// TIA Portal project "PROJEKT_PLC_PALIWKO" (V15.1)

(* hardware
DEVICE "S7-1200 station_1"  S7-1200 Station
   slot 0: "Rack_0"  S7-1200 Rack  Rack  V1.0
   slot 1: "PLC_1"  CPU 1212C AC/DC/Rly  6ES7 212-1BE40-0XB0  V4.2
DEVICE "HMI_1"  KTP700 Basic PN
   slot 0: "HMI_1"  KTP700 Basic PN  6AV2 123-2GB03-0AX0  15.0.0.0
   slot 1: "HMI_RT_1"  KTP700 Basic PN  6AV2 123-2GB03-0AX0  15.0.0.0
   slot 5: "HMI_1.IE_CP_1"  PROFINET Interface  15.0.0.0
      slot 1: "PROFINET Interface_1"  PROFINET Interface
         slot 1: "Port_1"  Port
*)

// ===== PLC "PLC_1"  CPU 1212C AC/DC/Rly =====

VAR_GLOBAL   // PLC tag table "Default tag table"
   "Adam" AT %M0.1 : Bool;
   "Ignacy" AT %M0.2 : Bool;
   "Kuba" AT %M0.3 : Bool;
   "Mateusz" AT %M0.4 : Bool;
   "Stachu" AT %M0.5 : Bool;
   "Limit_paliwa_adam" AT %M10.0 : Bool;
   "Limit_paliwa_ignacy" AT %M10.2 : Bool;
   "Limit_paliwa_kuba" AT %M10.3 : Bool;
   "Limit_paliwa_stachu" AT %M10.4 : Bool;
   "Limit_paliwa_mateusz" AT %M10.5 : Bool;
   "FuelingActive" AT %M10.6 : Bool;
   "Blokada_nalewania1" AT %M100.1 : Bool;
   "Blokada_nalewania2" AT %M100.2 : Bool;
   "Blokada_przelania_adam" AT %M4.0 : Bool;
   "Blokada_przelania_ignacy" AT %M4.1 : Bool;
   "Blokada_przelania_kuba" AT %M4.2 : Bool;
   "Blokada_przelania_mateusz" AT %M4.3 : Bool;
   "Blokada_przelania_stachu" AT %M4.4 : Bool;
END_VAR

TYPE "Kierowca"
   STRUCT
      Imie : String;
      Ilosc_Paliwa_Z : Int;
      Data_wydania : DTL;
   END_STRUCT;
END_TYPE

DATA_BLOCK "User_Data"   // DB1
{ S7_Optimized_Access := 'TRUE' }
VERSION : 0.1
   VAR
      Login : String;
      Adam : "Kierowca";
      Kuba : "Kierowca";
      Stachu : "Kierowca";
      Ignacy : "Kierowca";
      Mateusz : "Kierowca";
      Czy_Nalac : Bool;
      Done : Int;
   END_VAR
BEGIN
   Adam.Ilosc_Paliwa_Z := 200;
   Adam.Imie := 'Adam';
   Kuba.Imie := 'Kuba';
   Kuba.Ilosc_Paliwa_Z := 200;
   Stachu.Imie := 'Stachu';
   Stachu.Ilosc_Paliwa_Z := 200;
   Ignacy.Imie := 'Ignacy';
   Ignacy.Ilosc_Paliwa_Z := 200;
   Mateusz.Imie := 'Mateusz';
   Mateusz.Ilosc_Paliwa_Z := 200;
END_DATA_BLOCK

DATA_BLOCK "HMI"   // DB2
{ S7_Optimized_Access := 'TRUE' }
VERSION : 0.1
   VAR
      Current_User : String;
      Godzina : Time_Of_Day;
      Data : Date;
      Ile_Paliwa_z : Int;
      Ile_Paliwa_n : Int;
      Czy_nalac : Bool;
      Nalewanie_aktywne : Bool;
   END_VAR
BEGIN
END_DATA_BLOCK

DATA_BLOCK "Block_1_DB"   // DB3
{ S7_Optimized_Access := 'TRUE' }
VERSION : 0.1
// stored: InstanceOfName Block_1
"Block_1"
BEGIN
END_DATA_BLOCK

// folder: System blocks/Program resources

DATA_BLOCK "IEC_Timer_0_DB"   // DB5
{ S7_Optimized_Access := 'TRUE' }
AUTHOR : Simatic
FAMILY : IEC
NAME : IEC_TMR
VERSION : 1.0
// stored: InstanceOfName IEC_TIMER
"IEC_TIMER"
BEGIN
END_DATA_BLOCK

DATA_BLOCK "IEC_Timer_0_DB_1"   // DB6
{ S7_Optimized_Access := 'TRUE' }
AUTHOR : Simatic
FAMILY : IEC
NAME : IEC_TMR
VERSION : 1.0
// stored: InstanceOfName IEC_TIMER
"IEC_TIMER"
BEGIN
END_DATA_BLOCK

// folder: (top level)

FUNCTION_BLOCK "Block_1"   // FB1, LAD
TITLE = Pouring
{ S7_Optimized_Access := 'TRUE' }
VERSION : 0.1
// All the fuel dispensing logic happens
   VAR_TEMP   // added for the SCL form of the ladder/FBD networks
      _w1 : Bool;
   END_VAR
BEGIN

REGION Network 1: Trigger
   // Triggering the "pour" sequence
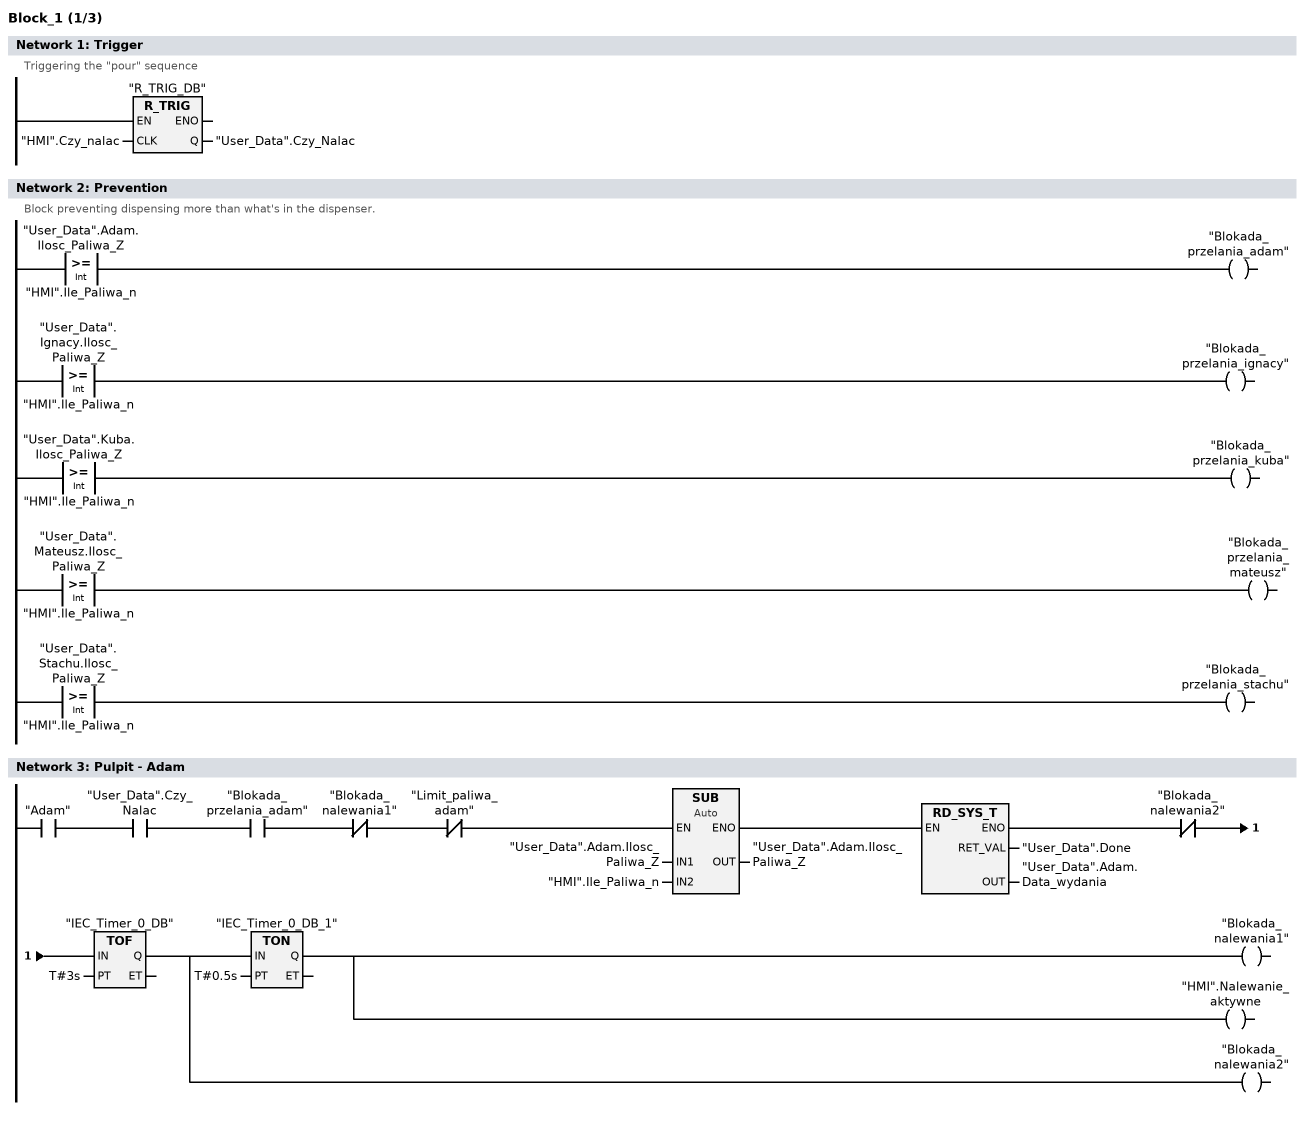
   "R_TRIG_DB"(CLK := "HMI".Czy_nalac, Q => "User_Data".Czy_Nalac);   // R_TRIG
END_REGION

REGION Network 2: Prevention
   // Block preventing dispensing more than what's in the dispenser.
   RUNG wire#powerrail
      { S7_Templates := "SrcType := Int" } GE_Contact(in1 := "User_Data".Adam.Ilosc_Paliwa_Z, in2 := "HMI".Ile_Paliwa_n)
      Coil( "Blokada_przelania_adam" )
   END_RUNG
   RUNG wire#powerrail
      { S7_Templates := "SrcType := Int" } GE_Contact(in1 := "User_Data".Ignacy.Ilosc_Paliwa_Z, in2 := "HMI".Ile_Paliwa_n)
      Coil( "Blokada_przelania_ignacy" )
   END_RUNG
   RUNG wire#powerrail
      { S7_Templates := "SrcType := Int" } GE_Contact(in1 := "User_Data".Kuba.Ilosc_Paliwa_Z, in2 := "HMI".Ile_Paliwa_n)
      Coil( "Blokada_przelania_kuba" )
   END_RUNG
   RUNG wire#powerrail
      { S7_Templates := "SrcType := Int" } GE_Contact(in1 := "User_Data".Mateusz.Ilosc_Paliwa_Z, in2 := "HMI".Ile_Paliwa_n)
      Coil( "Blokada_przelania_mateusz" )
   END_RUNG
   RUNG wire#powerrail
      { S7_Templates := "SrcType := Int" } GE_Contact(in1 := "User_Data".Stachu.Ilosc_Paliwa_Z, in2 := "HMI".Ile_Paliwa_n)
      Coil( "Blokada_przelania_stachu" )
   END_RUNG
   // the same network as SCL:
   "Blokada_przelania_adam" := "User_Data".Adam.Ilosc_Paliwa_Z >= "HMI".Ile_Paliwa_n;
   "Blokada_przelania_ignacy" := "User_Data".Ignacy.Ilosc_Paliwa_Z >= "HMI".Ile_Paliwa_n;
   "Blokada_przelania_kuba" := "User_Data".Kuba.Ilosc_Paliwa_Z >= "HMI".Ile_Paliwa_n;
   "Blokada_przelania_mateusz" := "User_Data".Mateusz.Ilosc_Paliwa_Z >= "HMI".Ile_Paliwa_n;
   "Blokada_przelania_stachu" := "User_Data".Stachu.Ilosc_Paliwa_Z >= "HMI".Ile_Paliwa_n;
END_REGION

REGION Network 3: Pulpit - Adam
   // ENO of a box is taken as its EN; it also drops when the box reports an error
   #_w1 := "Adam" AND "User_Data".Czy_Nalac AND "Blokada_przelania_adam" AND NOT "Blokada_nalewania1" AND NOT "Limit_paliwa_adam";
   IF #_w1 THEN
       "User_Data".Adam.Ilosc_Paliwa_Z := "User_Data".Adam.Ilosc_Paliwa_Z - "HMI".Ile_Paliwa_n;
       "User_Data".Done := RD_SYS_T(OUT => "User_Data".Adam.Data_wydania);
   END_IF;
   "IEC_Timer_0_DB".TOF(IN := #_w1 AND NOT "Blokada_nalewania2", PT := T#3s);
   "IEC_Timer_0_DB_1".TON(IN := "IEC_Timer_0_DB".Q, PT := T#0.5s);
   "Blokada_nalewania1" := "IEC_Timer_0_DB_1".Q;
   "HMI".Nalewanie_aktywne := "IEC_Timer_0_DB_1".Q;
   "Blokada_nalewania2" := "IEC_Timer_0_DB".Q;
END_REGION

REGION Network 4: Pulpit - Ignacy
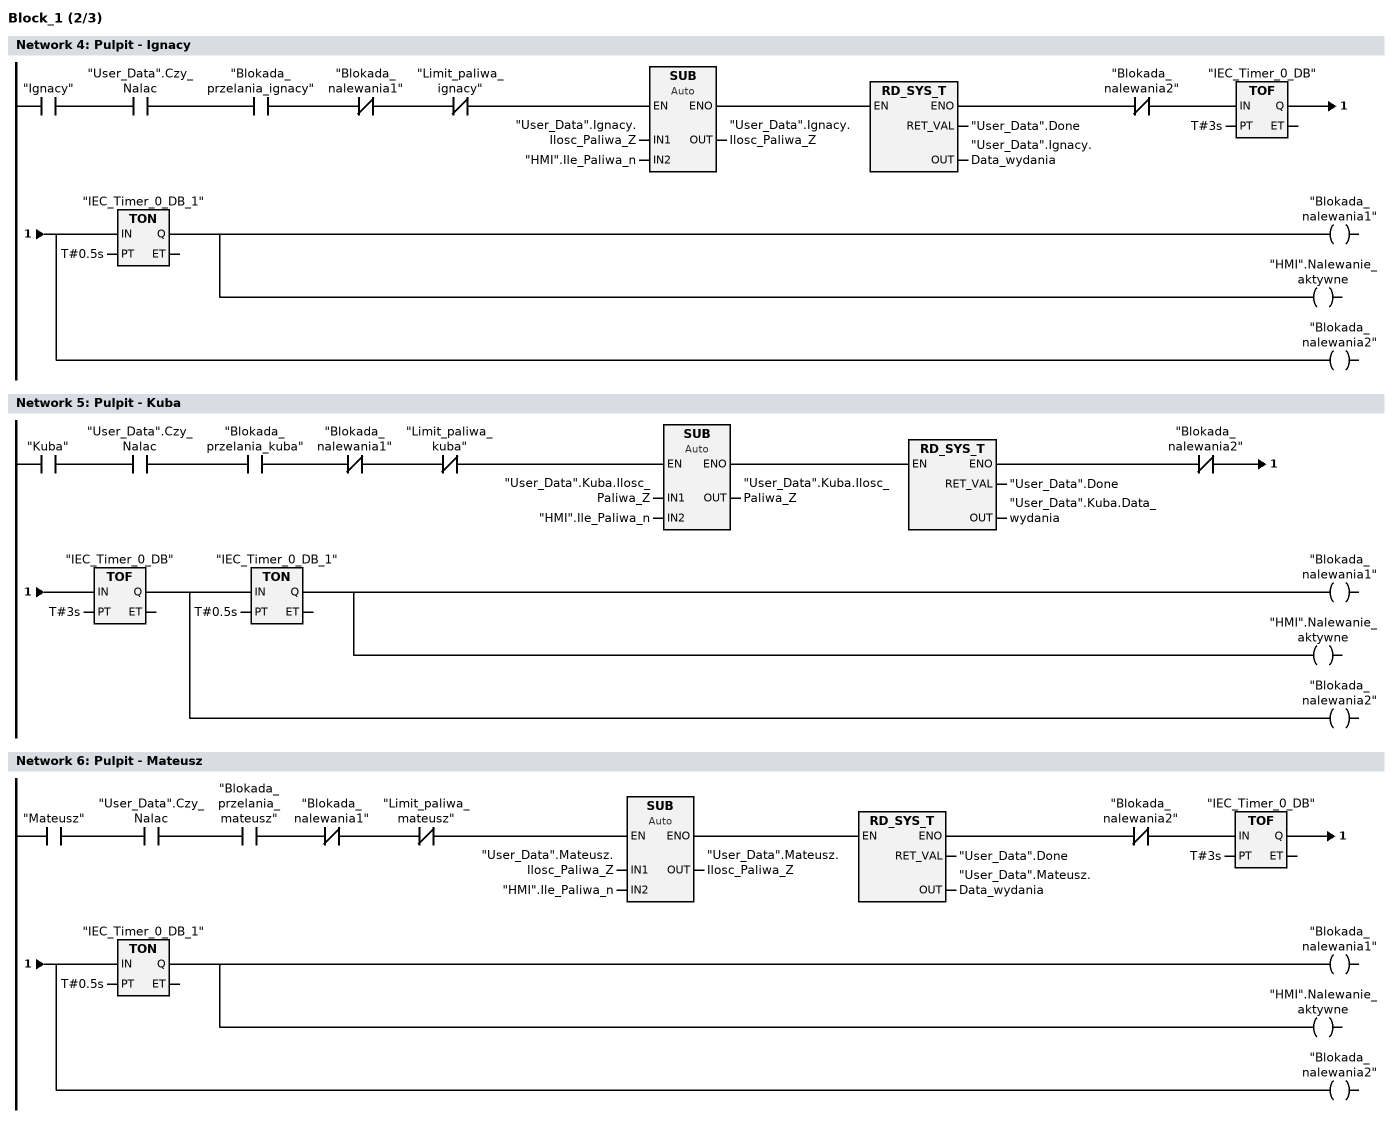
   // ENO of a box is taken as its EN; it also drops when the box reports an error
   #_w1 := "Ignacy" AND "User_Data".Czy_Nalac AND "Blokada_przelania_ignacy" AND NOT "Blokada_nalewania1" AND NOT "Limit_paliwa_ignacy";
   IF #_w1 THEN
       "User_Data".Ignacy.Ilosc_Paliwa_Z := "User_Data".Ignacy.Ilosc_Paliwa_Z - "HMI".Ile_Paliwa_n;
       "User_Data".Done := RD_SYS_T(OUT => "User_Data".Ignacy.Data_wydania);
   END_IF;
   "IEC_Timer_0_DB".TOF(IN := #_w1 AND NOT "Blokada_nalewania2", PT := T#3s);
   "IEC_Timer_0_DB_1".TON(IN := "IEC_Timer_0_DB".Q, PT := T#0.5s);
   "Blokada_nalewania1" := "IEC_Timer_0_DB_1".Q;
   "HMI".Nalewanie_aktywne := "IEC_Timer_0_DB_1".Q;
   "Blokada_nalewania2" := "IEC_Timer_0_DB".Q;
END_REGION

REGION Network 5: Pulpit - Kuba
   // ENO of a box is taken as its EN; it also drops when the box reports an error
   #_w1 := "Kuba" AND "User_Data".Czy_Nalac AND "Blokada_przelania_kuba" AND NOT "Blokada_nalewania1" AND NOT "Limit_paliwa_kuba";
   IF #_w1 THEN
       "User_Data".Kuba.Ilosc_Paliwa_Z := "User_Data".Kuba.Ilosc_Paliwa_Z - "HMI".Ile_Paliwa_n;
       "User_Data".Done := RD_SYS_T(OUT => "User_Data".Kuba.Data_wydania);
   END_IF;
   "IEC_Timer_0_DB".TOF(IN := #_w1 AND NOT "Blokada_nalewania2", PT := T#3s);
   "IEC_Timer_0_DB_1".TON(IN := "IEC_Timer_0_DB".Q, PT := T#0.5s);
   "Blokada_nalewania1" := "IEC_Timer_0_DB_1".Q;
   "HMI".Nalewanie_aktywne := "IEC_Timer_0_DB_1".Q;
   "Blokada_nalewania2" := "IEC_Timer_0_DB".Q;
END_REGION

REGION Network 6: Pulpit - Mateusz
   // ENO of a box is taken as its EN; it also drops when the box reports an error
   #_w1 := "Mateusz" AND "User_Data".Czy_Nalac AND "Blokada_przelania_mateusz" AND NOT "Blokada_nalewania1" AND NOT "Limit_paliwa_mateusz";
   IF #_w1 THEN
       "User_Data".Mateusz.Ilosc_Paliwa_Z := "User_Data".Mateusz.Ilosc_Paliwa_Z - "HMI".Ile_Paliwa_n;
       "User_Data".Done := RD_SYS_T(OUT => "User_Data".Mateusz.Data_wydania);
   END_IF;
   "IEC_Timer_0_DB".TOF(IN := #_w1 AND NOT "Blokada_nalewania2", PT := T#3s);
   "IEC_Timer_0_DB_1".TON(IN := "IEC_Timer_0_DB".Q, PT := T#0.5s);
   "Blokada_nalewania1" := "IEC_Timer_0_DB_1".Q;
   "HMI".Nalewanie_aktywne := "IEC_Timer_0_DB_1".Q;
   "Blokada_nalewania2" := "IEC_Timer_0_DB".Q;
END_REGION

REGION Network 7: Pulpit - Stachu
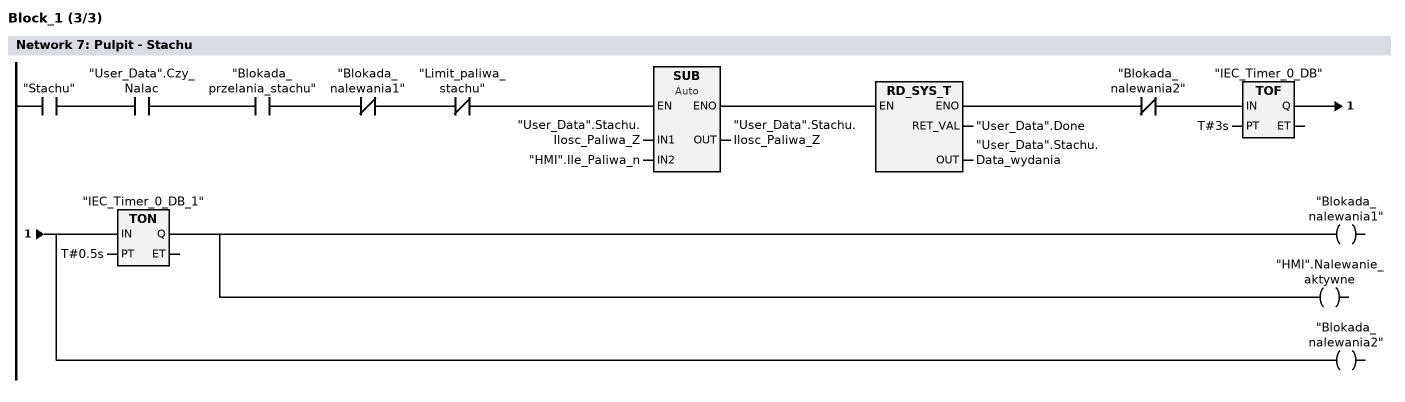
   // ENO of a box is taken as its EN; it also drops when the box reports an error
   #_w1 := "Stachu" AND "User_Data".Czy_Nalac AND "Blokada_przelania_stachu" AND NOT "Blokada_nalewania1" AND NOT "Limit_paliwa_stachu";
   IF #_w1 THEN
       "User_Data".Stachu.Ilosc_Paliwa_Z := "User_Data".Stachu.Ilosc_Paliwa_Z - "HMI".Ile_Paliwa_n;
       "User_Data".Done := RD_SYS_T(OUT => "User_Data".Stachu.Data_wydania);
   END_IF;
   "IEC_Timer_0_DB".TOF(IN := #_w1 AND NOT "Blokada_nalewania2", PT := T#3s);
   "IEC_Timer_0_DB_1".TON(IN := "IEC_Timer_0_DB".Q, PT := T#0.5s);
   "Blokada_nalewania1" := "IEC_Timer_0_DB_1".Q;
   "HMI".Nalewanie_aktywne := "IEC_Timer_0_DB_1".Q;
   "Blokada_nalewania2" := "IEC_Timer_0_DB".Q;
END_REGION
END_FUNCTION_BLOCK

ORGANIZATION_BLOCK "Main"   // OB1, LAD, ProgramCycle
TITLE = "Main Program Sweep (Cycle)"
{ S7_Optimized_Access := 'TRUE' }
VERSION : 0.1
BEGIN

REGION Network 1: User - data
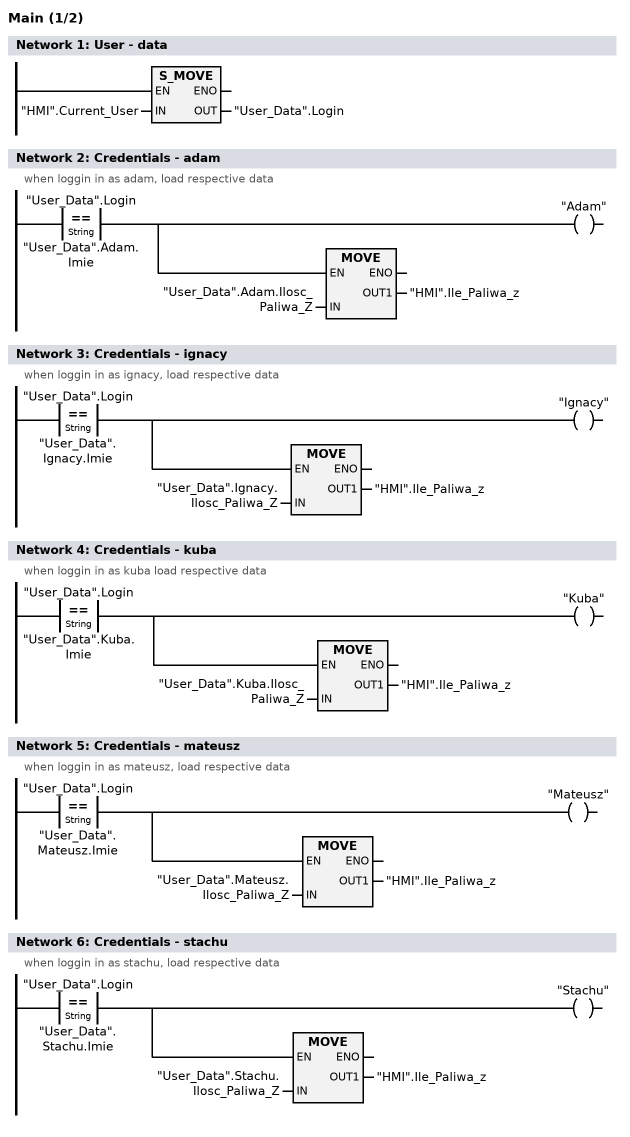
   RUNG wire#powerrail
      S_Move(in := "HMI".Current_User, out => "User_Data".Login)
   END_RUNG
   // the same network as SCL:
   "User_Data".Login := "HMI".Current_User;
END_REGION

REGION Network 2: Credentials - adam
   // when loggin in as adam, load respective data
   RUNG wire#powerrail
      { S7_Templates := "SrcType := String" } EQ_Contact(in1 := "User_Data".Login, in2 := "User_Data".Adam.Imie)
      wire#w1
      Coil( "Adam" )
   END_RUNG
   RUNG wire#w1
      Move(in := "User_Data".Adam.Ilosc_Paliwa_Z, out1 => "HMI".Ile_Paliwa_z)
   END_RUNG
   // the same network as SCL:
   "Adam" := "User_Data".Login = "User_Data".Adam.Imie;
   IF "Adam" THEN "HMI".Ile_Paliwa_z := "User_Data".Adam.Ilosc_Paliwa_Z; END_IF;
END_REGION

REGION Network 3: Credentials - ignacy
   // when loggin in as ignacy, load respective data
   RUNG wire#powerrail
      { S7_Templates := "SrcType := String" } EQ_Contact(in1 := "User_Data".Login, in2 := "User_Data".Ignacy.Imie)
      wire#w1
      Coil( "Ignacy" )
   END_RUNG
   RUNG wire#w1
      Move(in := "User_Data".Ignacy.Ilosc_Paliwa_Z, out1 => "HMI".Ile_Paliwa_z)
   END_RUNG
   // the same network as SCL:
   "Ignacy" := "User_Data".Login = "User_Data".Ignacy.Imie;
   IF "Ignacy" THEN "HMI".Ile_Paliwa_z := "User_Data".Ignacy.Ilosc_Paliwa_Z; END_IF;
END_REGION

REGION Network 4: Credentials - kuba
   // when loggin in as kuba load respective data
   RUNG wire#powerrail
      { S7_Templates := "SrcType := String" } EQ_Contact(in1 := "User_Data".Login, in2 := "User_Data".Kuba.Imie)
      wire#w1
      Coil( "Kuba" )
   END_RUNG
   RUNG wire#w1
      Move(in := "User_Data".Kuba.Ilosc_Paliwa_Z, out1 => "HMI".Ile_Paliwa_z)
   END_RUNG
   // the same network as SCL:
   "Kuba" := "User_Data".Login = "User_Data".Kuba.Imie;
   IF "Kuba" THEN "HMI".Ile_Paliwa_z := "User_Data".Kuba.Ilosc_Paliwa_Z; END_IF;
END_REGION

REGION Network 5: Credentials - mateusz
   // when loggin in as mateusz, load respective data
   RUNG wire#powerrail
      { S7_Templates := "SrcType := String" } EQ_Contact(in1 := "User_Data".Login, in2 := "User_Data".Mateusz.Imie)
      wire#w1
      Coil( "Mateusz" )
   END_RUNG
   RUNG wire#w1
      Move(in := "User_Data".Mateusz.Ilosc_Paliwa_Z, out1 => "HMI".Ile_Paliwa_z)
   END_RUNG
   // the same network as SCL:
   "Mateusz" := "User_Data".Login = "User_Data".Mateusz.Imie;
   IF "Mateusz" THEN "HMI".Ile_Paliwa_z := "User_Data".Mateusz.Ilosc_Paliwa_Z; END_IF;
END_REGION

REGION Network 6: Credentials - stachu
   // when loggin in as stachu, load respective data
   RUNG wire#powerrail
      { S7_Templates := "SrcType := String" } EQ_Contact(in1 := "User_Data".Login, in2 := "User_Data".Stachu.Imie)
      wire#w1
      Coil( "Stachu" )
   END_RUNG
   RUNG wire#w1
      Move(in := "User_Data".Stachu.Ilosc_Paliwa_Z, out1 => "HMI".Ile_Paliwa_z)
   END_RUNG
   // the same network as SCL:
   "Stachu" := "User_Data".Login = "User_Data".Stachu.Imie;
   IF "Stachu" THEN "HMI".Ile_Paliwa_z := "User_Data".Stachu.Ilosc_Paliwa_Z; END_IF;
END_REGION

REGION Network 7: Call FB1
   // FB1 - where all the fuel dispensing logic happens
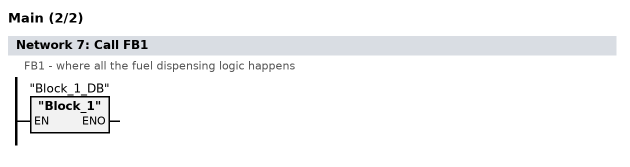
   RUNG wire#powerrail
      "Block_1_DB"()
   END_RUNG
   // the same network as SCL:
   "Block_1_DB"();   // "Block_1"
END_REGION
END_ORGANIZATION_BLOCK

(* ===== HMI "HMI_RT_1" =====
system functions are stored by id; their names below are inferred from use
connection "HMI_Connection_1": ETHERNET, SMART_S7_1200_OMS

HMI tags "Default tag table"
   "HMI_Current_User" : String[254] = PLC HMI.Current_User, 1 s
   "HMI_Ile_Paliwa_z" : Int = PLC HMI.Ile_Paliwa_z, 1 s
   "HMI_Ile_Paliwa_n" : Int = PLC HMI.Ile_Paliwa_n, 1 s
   "HMI_Czy_nalac" : Bool = PLC HMI.Czy_nalac, 1 s
   "HMI_Data_Godzina" : Time_Of_Day = PLC HMI.Godzina, 1 s
   "HMI_Data" : Date = PLC HMI.Data, 1 s
   "HMI_Nalewanie_aktywne" : Bool = PLC HMI.Nalewanie_aktywne AT %DB1.DBX0.0, 500 ms
   "FuelingActive" : Bool = PLC FuelingActive AT %M10.6, 1 s

Template "Template_1" 800x480
   Button "Alarms" at 512,428 size 71x50; TextOff 'Alarms / Alarm'; PictureOff "AlarmDisplay_KTP700_Basic_PN_TR"; PictureOn "AlarmDisplay_KTP700_Basic_PN_TR"
      on Release: function_ef3f5d25("Alarm window_Unacknowledged", -1)
   Button "Exit" at 411,428 size 71x50; TextOff 'Exit'; PictureOff "ExitRuntime_KTP700_Basic_PN_TR"; PictureOn "ExitRuntime_KTP700_Basic_PN_TR"
      on Release: StopRuntime(0)
   Button "Log on" at 311,428 size 71x50; TextOff 'Log on'; PictureOff "Login_KTP700_Basic_PN_TR"; PictureOn "Login_KTP700_Basic_PN_TR"
      on Release: function_a2a04561()
   Button "Start screen" at 211,428 size 71x50; TextOff 'Start screen / Ekran początkowy'; PictureOff "NavigateHome_KTP700_Basic_PN_TR"; PictureOn "NavigateHome_KTP700_Basic_PN_TR"
      on Release: ActivateScreen("Logowanie", 0)

screen "Logowanie" 800x480, template "Template_1"
   on GenerateScreen: function_f41c6f6c("HMI_Current_User")
   Button "Button_1" at 318,194 size 152x88; TextOff 'Log in / Zaloguj / Anmelden'; Authorization "Nalewanie"
      on Click: ActivateScreen("Nalewanie", 0)
   Button "Button_2" at 612,15 size 174x30; TextOff 'Change language / Zmień język / Sprache ändern'
      on Release: function_fb9197e8(-1)
   TextField "Text field_1" at 5,2 size 360x55; Text 'Electronic fuel distribution system / Elektroniczny system rozdzielni paliwa / Elektronisches Kraftstoffverteilungssystem'

screen "Nalewanie" 800x480
   on GenerateScreen: function_f41c6f6c("HMI_Current_User")
   Button "Button_1" at 615,390 size 135x56; TextOff 'Log out / Wyloguj / Abmelden'
      on Click: ActivateScreen("Logowanie", 0); function_f23ef4c9()
   IOField "I/O field_1" at 138,139 size 141x44; FormatPattern s99999
      ProcessValue <- "HMI_Ile_Paliwa_z"
   TextField "Text field_1" at 137,115 size 175x23; Text 'Distributor status / Stan dystrubutora / Status des Verteilers'
   IOField "I/O field_2" at 530,139 size 141x44; FormatPattern s99999
      ProcessValue <- "HMI_Ile_Paliwa_n"
   TextField "Text field_2" at 531,115 size 143x23; Text 'Dispensing order / Zlecenie rozlewu / Abfüllauftrag'
   Button "Button_2" at 343,244 size 122x53; TextOff 'Pour / Nalej / Einfüllen'
      on Press: SetBit("HMI_Czy_nalac"); function_fd9437ed(0, "Data_Godzina")
      on Release: ResetBit("HMI_Czy_nalac")
   DateTimeField "Date/time field_1" at 17,12 size 219x32
   TextField "Text field_3" at 530,204 size 141x23; Text 'Pouring... / Nalewanie... / Wird eingefüllt...'
      Visibility <- "HMI_Nalewanie_aktywne"
   Button "Button_3" at 612,15 size 174x30; TextOff 'Change language / Zmień język / Sprache ändern'
      on Release: function_fb9197e8(-1)
*)